KUKA KRL program: wkz6_com_01_st01_g01_ot2.src, wkz6_com_01_st01_g01_ot2.dat

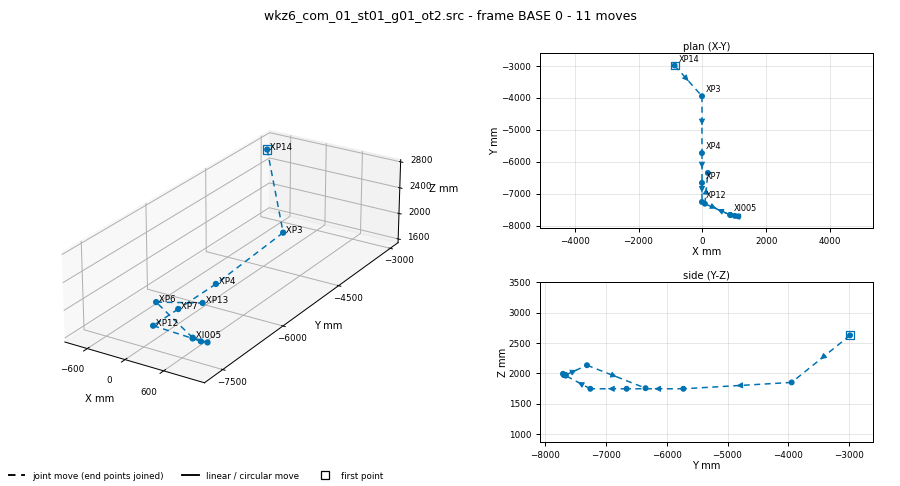
[picture p0: tool path of wkz6_com_01_st01_g01_ot2.src in frame BASE 0, 11 of 11 moves have a stored position in this frame; points joined in program order, loops and branches not executed]
--- wkz6_com_01_st01_g01_ot2.src ---
&ACCESS RVO1
&REL 10
&COMMENT Rolamento apoio geo LTBLTA
&PARAM DISKPATH = KRC:\R1\Program\MANIPULACAO NTC
&PARAM TEMPLATE = C:\KRC\Roboter\Template\vorgabe
&PARAM EDITMASK = *
DEF wkz6_com_01_st01_g01_ot2( )
;FOLD INI
  ;FOLD BASISTECH INI
    GLOBAL INTERRUPT DECL 3 WHEN $STOPMESS==TRUE DO IR_STOPM ( )
    INTERRUPT ON 3
    BAS (#INITMOV,0)
  ;ENDFOLD (BASISTECH INI)
;FOLD GRIPPERTECH INI
USER_GRP(0,DUMMY,DUMMY,GDEFAULT)
;ENDFOLD (GRIPPERTECH INI)
  ;FOLD USER INI
    ;Make your modifications here

  ;ENDFOLD (USER INI)
;ENDFOLD (INI)

; Caracterizacao dos meios de producao
; Changes: Posiciona Rolete na Traseira
; Modelos: Axor/Atego - LTB - LTA
; Versao Atual: 18/05/2017
; Name: P13.050-R3

chk_w6_wechs_ok ( )     ; CHECK GRIPPER AXOR/ATEGO

;FOLD PTP P14 CONT Vel=100 % PDAT13 Tool[6]:Gripper G0100R Base[0];%{PE}%R 8.2.20,%MKUKATPBASIS,%CMOVE,%VPTP,%P 1:PTP, 2:P14, 3:C_DIS, 5:100, 7:PDAT13
$BWDSTART=FALSE
PDAT_ACT=PPDAT13
FDAT_ACT=FP14
BAS(#PTP_PARAMS,100)
PTP XP14 C_DIS
;ENDFOLD
;FOLD PTP P3 CONT Vel=100 % PDAT5 Tool[6]:Gripper G0100R Base[0];%{PE}%R 8.2.20,%MKUKATPBASIS,%CMOVE,%VPTP,%P 1:PTP, 2:P3, 3:C_DIS, 5:100, 7:PDAT5
$BWDSTART=FALSE
PDAT_ACT=PPDAT5
FDAT_ACT=FP3
BAS(#PTP_PARAMS,100)
PTP XP3 C_DIS
;ENDFOLD

; ABRE GRAMPO Z7.1/2
;FOLD SET Z7.1/2 GRP AXOR State=OPN CONT at START Delay=1 ms;%{PE}%R 8.2.1,%MKUKATPGRP,%CGRP,%VGRP,%P 2:15, 4:1, 5:#YES, 6:GDAT26, 8:0, 10:1
TRIGGER WHEN DISTANCE=0 DELAY=1 DO H50(GRP_APO,15,1,GCONT) PRIO=-1
;ENDFOLD

;FOLD PTP P4 CONT Vel=100 % PDAT6 Tool[6]:Gripper G0100R Base[0];%{PE}%R 8.2.20,%MKUKATPBASIS,%CMOVE,%VPTP,%P 1:PTP, 2:P4, 3:C_DIS, 5:100, 7:PDAT6
$BWDSTART=FALSE
PDAT_ACT=PPDAT6
FDAT_ACT=FP4
BAS(#PTP_PARAMS,100)
PTP XP4 C_DIS
;ENDFOLD

;FOLD PTP P7 CONT Vel=100 % PDAT7 Tool[6]:Gripper G0100R Base[0];%{PE}%R 8.2.20,%MKUKATPBASIS,%CMOVE,%VPTP,%P 1:PTP, 2:P7, 3:C_DIS, 5:100, 7:PDAT7
$BWDSTART=FALSE
PDAT_ACT=PPDAT7
FDAT_ACT=FP7
BAS(#PTP_PARAMS,100)
PTP XP7 C_DIS
;ENDFOLD
; AGUARDA LIBERACAO PARA PRE_DEPOSITO
;FOLD OUT 3372 'Lib. pré Dep. Axor/Atego' State=TRUE ;%{PE}%R 8.2.20,%MKUKATPBASIS,%COUT,%VOUTX,%P 2:3372, 3:Lib. pré Dep. Axor/Atego, 5:TRUE, 6:
$OUT[3372]=TRUE
;ENDFOLD
;FOLD WAIT FOR ( IN 3372 'Lib. pré Deposito Axor/Atego' );%{PE}%R 8.2.20,%MKUKATPBASIS,%CEXT_WAIT_FOR,%VEXT_WAIT_FOR,%P 2:, 4:, 5:$IN, 6:3372, 7:Lib. pré Deposito Axor/Atego, 9:
WAIT FOR  ( $IN[3372] )
;ENDFOLD
;FOLD OUT 3372 'Lib. pré Dep. Axor/Atego' State=FALSE ;%{PE}%R 8.2.20,%MKUKATPBASIS,%COUT,%VOUTX,%P 2:3372, 3:Lib. pré Dep. Axor/Atego, 5:FALSE, 6:
$OUT[3372]=FALSE
;ENDFOLD
;FOLD OUT 3340 'Area_clear_AGV' State=FALSE ;%{PE}%R 8.2.20,%MKUKATPBASIS,%COUT,%VOUTX,%P 2:3340, 3:Area_clear_AGV, 5:FALSE, 6:
$OUT[3340]=FALSE
;ENDFOLD
;FOLD OUT 3348 'Fora area GEOBOX' State=FALSE ;%{PE}%R 8.2.20,%MKUKATPBASIS,%COUT,%VOUTX,%P 2:3348, 3:Fora area GEOBOX, 5:FALSE, 6:
$OUT[3348]=FALSE
;ENDFOLD

;FOLD ; LIGA INTERTRAVAMENTO 1 C/ R1 NA PEGA DA GARRA 913;%{PE}%R 8.2.20,%MKUKATPBASIS,%CCOMMENT,%VNORMAL,%P 2:LIGA INTERTRAVAMENTO  1 C/ R1 NA PEGA DA GARRA 913
;ENDFOLD
;FOLD Collision.Monitoring_1_On ;%{PE}%MKUKATPUSER
COLLSTOP( 1, 1 ) ;Interrupt-Controlled
;ENDFOLD

; VERIFICA GRAMPO Z7.1/2 ABERTO
chk_w6_grp7_opn( )

;FOLD PTP P12 CONT Vel=100 % PDAT11 Tool[6]:Gripper G0100R Base[0];%{PE}%R 8.2.20,%MKUKATPBASIS,%CMOVE,%VPTP,%P 1:PTP, 2:P12, 3:C_DIS, 5:100, 7:PDAT11
$BWDSTART=FALSE
PDAT_ACT=PPDAT11
FDAT_ACT=FP12
BAS(#PTP_PARAMS,100)
PTP XP12 C_DIS
;ENDFOLD
;FOLD PTP l005 CONT Vel=100 % P_OLP2 Tool[6]:Gripper G0100R Base[0];%{PE}%R 8.2.20,%MKUKATPBASIS,%CMOVE,%VPTP,%P 1:PTP, 2:l005, 3:C_DIS, 5:100, 7:P_OLP2
$BWDSTART=FALSE
PDAT_ACT=PP_OLP2
FDAT_ACT=Fl005
BAS(#PTP_PARAMS,100)
PTP Xl005 C_DIS
;ENDFOLD
;FOLD LIN l020 CONT Vel=1 m/s CPDAT4 Tool[6]:Gripper G0100R Base[0];%{PE}%R 8.2.20,%MKUKATPBASIS,%CMOVE,%VLIN,%P 1:LIN, 2:l020, 3:C_DIS C_DIS, 5:1, 7:CPDAT4
$BWDSTART=FALSE
LDAT_ACT=LCPDAT4
FDAT_ACT=Fl020
BAS(#CP_PARAMS,1)
LIN Xl020 C_DIS C_DIS
;ENDFOLD

;FOLD ; ROLAMENTO POSICIONADO;%{PE}%R 8.2.20,%MKUKATPBASIS,%CCOMMENT,%VNORMAL,%P 2:ROLAMENTO  POSICIONADO
;ENDFOLD
;FOLD LIN l026 Vel=0.25 m/s CPDAT0 Tool[6]:Gripper G0100R Base[0];%{PE}%R 8.2.20,%MKUKATPBASIS,%CMOVE,%VLIN,%P 1:LIN, 2:l026, 3:, 5:0.25, 7:CPDAT0
$BWDSTART=FALSE
LDAT_ACT=LCPDAT0
FDAT_ACT=Fl026
BAS(#CP_PARAMS,0.25)
LIN Xl026
;ENDFOLD

; AGUARDA LIBERACAO PARA SAIDA DO APOIO
;FOLD OUT 3373 'Em pos de apoio axor atego' State=TRUE ;%{PE}%R 8.2.20,%MKUKATPBASIS,%COUT,%VOUTX,%P 2:3373, 3:Em pos de apoio axor atego, 5:TRUE, 6:
$OUT[3373]=TRUE
;ENDFOLD
;FOLD WAIT FOR ( IN 3373 'Lib Sair do apoio rolete geo axor atego' );%{PE}%R 8.2.20,%MKUKATPBASIS,%CEXT_WAIT_FOR,%VEXT_WAIT_FOR,%P 2:, 4:, 5:$IN, 6:3373, 7:Lib Sair do apoio rolete geo axor atego, 9:
WAIT FOR  ( $IN[3373] )
;ENDFOLD
;FOLD OUT 3373 'Em pos de apoio axor atego' State=FALSE ;%{PE}%R 8.2.20,%MKUKATPBASIS,%COUT,%VOUTX,%P 2:3373, 3:Em pos de apoio axor atego, 5:FALSE, 6:
$OUT[3373]=FALSE
;ENDFOLD

;FOLD LIN l030 CONT Vel=2 m/s CPDAT5 Tool[6]:Gripper G0100R Base[0];%{PE}%R 8.2.20,%MKUKATPBASIS,%CMOVE,%VLIN,%P 1:LIN, 2:l030, 3:C_DIS C_DIS, 5:2, 7:CPDAT5
$BWDSTART=FALSE
LDAT_ACT=LCPDAT5
FDAT_ACT=Fl030
BAS(#CP_PARAMS,2)
LIN Xl030 C_DIS C_DIS
;ENDFOLD
;FOLD PTP P6 CONT Vel=100 % PDAT4 Tool[6]:Gripper G0100R Base[0];%{PE}%R 8.2.20,%MKUKATPBASIS,%CMOVE,%VPTP,%P 1:PTP, 2:P6, 3:C_DIS, 5:100, 7:PDAT4
$BWDSTART=FALSE
PDAT_ACT=PPDAT4
FDAT_ACT=FP6
BAS(#PTP_PARAMS,100)
PTP XP6 C_DIS
;ENDFOLD
;FOLD PTP P13 CONT Vel=100 % PDAT12 Tool[6]:Gripper G0100R Base[0];%{PE}%R 8.2.20,%MKUKATPBASIS,%CMOVE,%VPTP,%P 1:PTP, 2:P13, 3:C_DIS, 5:100, 7:PDAT12
$BWDSTART=FALSE
PDAT_ACT=PPDAT12
FDAT_ACT=FP13
BAS(#PTP_PARAMS,100)
PTP XP13 C_DIS
;ENDFOLD

END

--- wkz6_com_01_st01_g01_ot2.dat ---
&ACCESS RVO1
&REL 10
&COMMENT Rolamento apoio geo LTBLTA
&PARAM DISKPATH = KRC:\R1\Program\MANIPULACAO NTC
&PARAM TEMPLATE = C:\KRC\Roboter\Template\vorgabe
&PARAM EDITMASK = *
DEFDAT  wkz6_com_01_st01_g01_ot2
;FOLD EXTERNAL DECLARATIONS;%{PE}%MKUKATPBASIS,%CEXT,%VCOMMON,%P
;FOLD GRIPPERTECH EXT
EXT  H50 (INT  :IN,INT  :IN,INT  :IN,GRP_TYP  :IN )
;ENDFOLD (GRIPPERTECH EXT)
;FOLD SPOTTECH EXT

;ENDFOLD (SPOTTECH EXT)
;FOLD BASISTECH EXT;%{PE}%MKUKATPBASIS,%CEXT,%VEXT,%P
EXT  BAS (BAS_COMMAND  :IN,REAL  :IN )
DECL INT SUCCESS
;ENDFOLD (BASISTECH EXT)
;FOLD USER EXT;%{E}%MKUKATPUSER,%CEXT,%VEXT,%P

;ENDFOLD (USER EXT)
;ENDFOLD (EXTERNAL DECLARATIONS)
DECL FDAT Fl005={TOOL_NO 6,BASE_NO 0,IPO_FRAME #BASE,POINT2[] " ",TQ_STATE FALSE}
DECL PDAT PP_OLP2={VEL 100.0,ACC 100.0,APO_DIST 30.0,APO_MODE #CDIS}
DECL E6POS Xl005={X 874.661377,Y -7665.34082,Z 1964.0,A -81.3817673,B -88.3855591,C -112.569397,S 2,T 35,E1 5000.0,E2 0.0,E3 0.0,E4 0.0,E5 0.0,E6 0.0}
DECL FDAT Fl010={TOOL_NO 6,BASE_NO 0,IPO_FRAME #BASE,POINT2[] " ",TQ_STATE FALSE}
DECL PDAT PP_OLP3={VEL 100.0,ACC 100.0,APO_DIST 30.0,APO_MODE #CDIS}
DECL E6POS Xl010={X 245.965103,Y -6431.59912,Z 1863.31104,A 159.308304,B -77.2926636,C -26.9483795,S 2,T 3,E1 3968.33398,E2 0.0,E3 0.0,E4 0.0,E5 0.0,E6 0.0}
DECL FDAT Fl020={TOOL_NO 6,BASE_NO 0,IPO_FRAME #BASE,POINT2[] " "}
DECL E6POS Xl020={X 1018.99597,Y -7695.07178,Z 1972.91394,A -130.374496,B -88.8259735,C -63.5509682,S 2,T 35,E1 5000.0,E2 0.0,E3 0.0,E4 0.0,E5 0.0,E6 0.0}
DECL FDAT Fl025={TOOL_NO 6,BASE_NO 0,IPO_FRAME #BASE,POINT2[] " "}
DECL E6POS Xl025={X 1115.22095,Y -7714.89209,Z 1978.854,A -163.379898,B -88.5089493,C -30.5284691,S 2,T 35,E1 5000.00098,E2 0.0,E3 0.0,E4 0.0,E5 0.0,E6 0.0}
DECL FDAT Fl030={TOOL_NO 6,BASE_NO 0,IPO_FRAME #BASE,POINT2[] " "}
DECL E6POS Xl030={X 874.655823,Y -7665.34619,Z 1974.60901,A -81.3771286,B -88.3856506,C -112.574303,S 6,T 59,E1 5000.0,E2 0.0,E3 0.0,E4 0.0,E5 0.0,E6 0.0}
DECL BASIS_SUGG_T LAST_BASIS={POINT1[] "P7                      ",POINT2[] "P7                      ",CP_PARAMS[] "CPDAT0                  ",PTP_PARAMS[] "PDAT7                   ",CONT[] "C_DIS                   ",CP_VEL[] "0.25                    ",PTP_VEL[] "100                     ",SYNC_PARAMS[] "SYNCDAT                 ",SPL_NAME[] "S0                      "}
DECL GRP_SUGG_T LAST_GRP={NUMBER[] "9                       ",STATE[] "2                       ",PARAMS[] "GDAT22                  "}
DECL GRP_TYP GGDAT2={G_APO #NO,GRP_TIME 0.200000003,CTRL #OFF,DLY 0,DST 1}
DECL GRP_TYP GGDAT1={G_APO #NO,GRP_TIME 0.200000003,CTRL #OFF,DLY 0,DST 1}
DECL GRP_TYP GGDAT3={G_APO #NO,GRP_TIME 0.200000003,CTRL #OFF,DLY 0,DST 1}
DECL GRP_TYP GGDAT4={G_APO #NO,GRP_TIME 0.200000003,CTRL #OFF,DLY 0,DST 1}
DECL GRP_TYP GGDAT5={G_APO #NO,GRP_TIME 0.200000003,CTRL #OFF,DLY 0,DST 1}
DECL GRP_TYP GGDAT6={G_APO #NO,GRP_TIME 0.200000003,CTRL #OFF,DLY 0,DST 1}
DECL GRP_TYP GGDAT7={G_APO #NO,GRP_TIME 0.200000003,CTRL #OFF,DLY 0,DST 1}
DECL GRP_TYP GGDAT8={G_APO #NO,GRP_TIME 0.200000003,CTRL #OFF,DLY 0,DST 1}
DECL GRP_TYP GGDAT9={G_APO #NO,GRP_TIME 0.200000003,CTRL #OFF,DLY 0,DST 1}
DECL GRP_TYP GGDAT10={G_APO #NO,GRP_TIME 0.200000003,CTRL #OFF,DLY 0,DST 1}
DECL GRP_TYP GGDAT11={G_APO #NO,GRP_TIME 0.200000003,CTRL #OFF,DLY 0,DST 1}
DECL GRP_TYP GGDAT12={G_APO #NO,GRP_TIME 0.200000003,CTRL #OFF,DLY 0,DST 1}
DECL GRP_TYP GGDAT13={G_APO #NO,GRP_TIME 0.200000003,CTRL #OFF,DLY 0,DST 1}
DECL GRP_TYP GGDAT14={G_APO #NO,GRP_TIME 0.200000003,CTRL #OFF,DLY 0,DST 1}
DECL GRP_TYP GGDAT15={G_APO #NO,GRP_TIME 0.200000003,CTRL #OFF,DLY 0,DST 1}
DECL GRP_TYP GGDAT16={G_APO #NO,GRP_TIME 0.200000003,CTRL #OFF,DLY 0,DST 1}
DECL GRP_TYP GGDAT17={G_APO #NO,GRP_TIME 0.200000003,CTRL #OFF,DLY 0,DST 1}
DECL GRP_TYP GGDAT18={G_APO #NO,GRP_TIME 0.200000003,CTRL #OFF,DLY 0,DST 1}
DECL E6POS XP5={X -12.1998396,Y -5726.93115,Z 1747.21899,A 162.530701,B -81.9720612,C -45.6247482,S 2,T 35,E1 3391.98511,E2 0.0,E3 0.0,E4 0.0,E5 0.0,E6 0.0}
DECL FDAT FP5={TOOL_NO 6,BASE_NO 0,IPO_FRAME #BASE,POINT2[] " ",TQ_STATE FALSE}
DECL PDAT PPDAT3={VEL 100.0,ACC 100.0,APO_DIST 100.0,APO_MODE #CDIS}
DECL GRP_TYP GGDAT19={G_APO #NO,GRP_TIME 0.200000003,CTRL #OFF,DLY 0,DST 1}
DECL LDAT LCPDAT3={VEL 2.0,ACC 100.0,APO_DIST 20.0,APO_FAC 50.0,AXIS_VEL 100.0,AXIS_ACC 100.0,ORI_TYP #VAR,CIRC_TYP #BASE,JERK_FAC 50.0,GEAR_JERK 50.0,EXAX_IGN 0}
DECL E6POS XP6={X 79.065712,Y -7314.14209,Z 2135.34399,A -55.6808586,B -84.730217,C -156.120605,S 2,T 35,E1 4464.73291,E2 0.0,E3 0.0,E4 0.0,E5 0.0,E6 0.0}
DECL FDAT FP6={TOOL_NO 6,BASE_NO 0,IPO_FRAME #BASE,POINT2[] " ",TQ_STATE FALSE}
DECL PDAT PPDAT4={VEL 100.0,ACC 100.0,APO_DIST 50.0,APO_MODE #CDIS}
DECL GRP_TYP GGDAT20={G_APO #NO,GRP_TIME 0.200000003,CTRL #OFF,DLY 0,DST 1}
DECL GRP_TYP GGDAT21={G_APO #NO,GRP_TIME 0.200000003,CTRL #OFF,DLY 0,DST 1}
DECL GRP_TYP GGDAT22={G_APO #NO,GRP_TIME 0.200000003,CTRL #OFF,DLY 0,DST 1}
DECL GRP_TYP GGDAT23={G_APO #NO,GRP_TIME 0.200000003,CTRL #OFF,DLY 0,DST 1}
DECL GRP_TYP GGDAT24={G_APO #NO,GRP_TIME 0.200000003,CTRL #OFF,DLY 0,DST 1}
DECL GRP_TYP GGDAT25={G_APO #NO,GRP_TIME 0.200000003,CTRL #OFF,DLY 0,DST 1}
DECL LDAT LCPDAT4={VEL 2.0,ACC 100.0,APO_DIST 50.0,APO_FAC 50.0,AXIS_VEL 100.0,AXIS_ACC 100.0,ORI_TYP #VAR,CIRC_TYP #BASE,JERK_FAC 50.0,GEAR_JERK 50.0,EXAX_IGN 0}
DECL LDAT LCPDAT5={VEL 2.0,ACC 100.0,APO_DIST 50.0,APO_FAC 50.0,AXIS_VEL 100.0,AXIS_ACC 100.0,ORI_TYP #VAR,CIRC_TYP #BASE,JERK_FAC 50.0,GEAR_JERK 50.0,EXAX_IGN 0}
DECL PDAT PPDAT11={VEL 100.0,ACC 100.0,APO_DIST 100.0,APO_MODE #CDIS}
DECL E6POS XP12={X -12.1998196,Y -7259.36914,Z 1747.21497,A 162.531204,B -81.9723892,C -45.6250801,S 2,T 35,E1 4924.42383,E2 0.0,E3 0.0,E4 0.0,E5 0.0,E6 0.0}
DECL FDAT FP12={TOOL_NO 6,BASE_NO 0,IPO_FRAME #BASE,POINT2[] " ",TQ_STATE FALSE}
DECL E6POS XP13={X 173.678406,Y -6349.35107,Z 1757.08997,A -27.3708801,B -75.7155533,C -130.396393,S 6,T 51,E1 4424.18994,E2 0.0,E3 0.0,E4 0.0,E5 0.0,E6 0.0}
DECL FDAT FP13={TOOL_NO 6,BASE_NO 0,IPO_FRAME #BASE,POINT2[] " ",TQ_STATE FALSE}
DECL PDAT PPDAT12={VEL 100.0,ACC 100.0,APO_DIST 100.0,APO_MODE #CDIS}
DECL E6POS XP14={X -867.852112,Y -2982.84692,Z 2626.92896,A 62.2299194,B 89.9792862,C -82.8014297,S 2,T 35,E1 1550.0,E2 0.0,E3 0.0,E4 0.0,E5 0.0,E6 0.0}
DECL FDAT FP14={TOOL_NO 6,BASE_NO 0,IPO_FRAME #BASE,POINT2[] " ",TQ_STATE FALSE}
DECL PDAT PPDAT13={VEL 100.0,ACC 100.0,APO_DIST 100.0,APO_MODE #CDIS}
DECL GRP_TYP GCONT={G_APO #YES,GRP_TIME 0.0,CTRL #OFF,DLY 0,DST 0}
DECL E6POS XP15={X -95.3618698,Y -3880.63892,Z 1742.48096,A -101.964798,B -88.8884735,C -143.026901,S 2,T 3,E1 1550.01001,E2 0.0,E3 0.0,E4 0.0,E5 0.0,E6 0.0}
DECL FDAT FP15={TOOL_NO 6,BASE_NO 0,IPO_FRAME #BASE,POINT2[] " ",TQ_STATE FALSE}
DECL PDAT PPDAT14={VEL 100.0,ACC 100.0,APO_DIST 50.0,APO_MODE #CDIS}
DECL E6POS XP1={X 261.918915,Y -7112.47021,Z 1918.13904,A 156.110901,B -72.7941437,C -23.8569393,S 2,T 3,E1 4636.14209,E2 0.0,E3 0.0,E4 0.0,E5 0.0,E6 0.0}
DECL FDAT FP1={TOOL_NO 6,BASE_NO 0,IPO_FRAME #BASE,POINT2[] " ",TQ_STATE FALSE}
DECL PDAT PPDAT1={VEL 100.0,ACC 100.0,APO_DIST 100.0,APO_MODE #CDIS}
DECL E6POS XP2={X 824.372498,Y -7588.68604,Z 1964.00305,A -81.3776321,B -88.3856964,C -112.573601,S 2,T 3,E1 5000.0,E2 0.0,E3 0.0,E4 0.0,E5 0.0,E6 0.0}
DECL FDAT FP2={TOOL_NO 6,BASE_NO 0,IPO_FRAME #BASE,POINT2[] " ",TQ_STATE FALSE}
DECL PDAT PPDAT2={VEL 100.0,ACC 100.0,APO_DIST 100.0,APO_MODE #CDIS}
DECL PDAT PPDAT0={VEL 100.0,ACC 100.0,APO_DIST 100.0,APO_MODE #CDIS}
DECL E6POS XP0={X 173.678894,Y -6349.34717,Z 1757.09302,A -27.3723507,B -75.7156067,C -130.394806,S 6,T 51,E1 4424.19189,E2 0.0,E3 0.0,E4 0.0,E5 0.0,E6 0.0}
DECL FDAT FP0={TOOL_NO 6,BASE_NO 0,IPO_FRAME #BASE,POINT2[] " ",TQ_STATE FALSE}
DECL LDAT LCPDAT1={VEL 2.0,ACC 100.0,APO_DIST 100.0,APO_FAC 50.0,AXIS_VEL 100.0,AXIS_ACC 100.0,ORI_TYP #VAR,CIRC_TYP #BASE,JERK_FAC 50.0,GEAR_JERK 50.0,EXAX_IGN 0}
DECL E6POS XP3={X -10.7895098,Y -3944.25708,Z 1851.89294,A 143.863602,B -81.0644226,C -26.6961403,S 2,T 35,E1 1550.00098,E2 0.0,E3 0.0,E4 0.0,E5 0.0,E6 0.0}
DECL FDAT FP3={TOOL_NO 6,BASE_NO 0,IPO_FRAME #BASE,POINT2[] " ",TQ_STATE FALSE}
DECL PDAT PPDAT5={VEL 100.0,ACC 100.0,APO_DIST 100.0,APO_MODE #CDIS}
DECL E6POS XP4={X -12.1995096,Y -5726.93115,Z 1747.21802,A 162.530396,B -81.9723969,C -45.6242905,S 2,T 35,E1 3391.98511,E2 0.0,E3 0.0,E4 0.0,E5 0.0,E6 0.0}
DECL FDAT FP4={TOOL_NO 6,BASE_NO 0,IPO_FRAME #BASE,POINT2[] " ",TQ_STATE FALSE}
DECL PDAT PPDAT6={VEL 100.0,ACC 100.0,APO_DIST 100.0,APO_MODE #CDIS}
DECL E6POS XP7={X -12.1997604,Y -6661.33496,Z 1747.21106,A 162.532104,B -81.9724274,C -45.6260109,S 2,T 35,E1 4326.39209,E2 0.0,E3 0.0,E4 0.0,E5 0.0,E6 0.0}
DECL FDAT FP7={TOOL_NO 6,BASE_NO 0,IPO_FRAME #BASE,POINT2[] " ",TQ_STATE FALSE}
DECL PDAT PPDAT7={VEL 100.0,ACC 100.0,APO_DIST 100.0,APO_MODE #CDIS}
DECL LDAT LCPDAT0={VEL 2.0,ACC 100.0,APO_DIST 20.0,APO_FAC 50.0,AXIS_VEL 100.0,AXIS_ACC 100.0,ORI_TYP #VAR,CIRC_TYP #BASE,JERK_FAC 50.0,GEAR_JERK 50.0,EXAX_IGN 0}
DECL E6POS Xl026={X 1128.51099,Y -7709.67822,Z 1993.271,A -130.332504,B -88.8254089,C -63.5924911,S 2,T 35,E1 5000.00391,E2 0.0,E3 0.0,E4 0.0,E5 0.0,E6 0.0}
DECL FDAT Fl026={TOOL_NO 6,BASE_NO 0,IPO_FRAME #BASE,POINT2[] " "}
ENDDAT
